FUNCTION_BLOCK WrappedComponentExample EXTENDS TcoCore.TcoComponent


VAR_OUTPUT
END_VAR
VAR
	_config:WrappedComponentExample_Config;
	_status:WrappedComponentExample_Status;
	_control:WrappedComponentExample_Control;
    _components:WrappedComponentsExample:= (Parent := THIS^);
	_throwTask:TcoCore.TcoTask(THIS^);
	_restoreTask:TcoCore.TcoTask(THIS^);

END_VAR

_throwTask();
_restoreTask.Enabled:=true;
_restoreTask();

PROPERTY Components : REFERENCE TO WrappedComponentsExample
GET
Components ref=_components;
END_GET
END_PROPERTY

(*~
	<docu>
		<summary>
			Restores this instance to the Ready state. Can be called explicitly or from within one of the restore mechanisms.	
		</summary>			
	</docu>	
~*)
METHOD  Restore : ITcoRestorable
END_METHOD

(*~
	<docu>
		<summary>
		    Custom service (manual, maintenance) logic.
			This method must be implemented in derived class.
		</summary>			
	</docu>	
~*)
METHOD PROTECTED  ServiceMode
END_METHOD

END_FUNCTION_BLOCK

(* stored: Version 1.1.0.1
   POU WrappedComponentExample: Id {bb4def30-cbc6-46bb-9bcc-fe384c9d62a8}, SpecialFunc None
   Property Components: Id {bda82270-6e27-4cda-be57-6208b70f70ff}
   Get Get: Id {4373dc8d-89bd-4ec1-ae7b-02b4f8528f42}
   Method Restore: Id {a8f20a69-5727-4e62-b0f2-8a099ded8a50}
   Method ServiceMode: Id {ed721f5f-f140-42d8-a720-a5e55b05821e} *)
